// Brief: Master Arm Standby
FUNCTION_BLOCK PUBLIC FB_StateCtrlPanelReady EXTENDS FB_SlaveArmCtrlBase
VAR_INPUT
END_VAR
VAR_OUTPUT
END_VAR
VAR
END_VAR

END_FUNCTION_BLOCK

(* stored: Version 1.1.0.1, ProductVersion 3.1.4024.12
   POU FB_StateCtrlPanelReady: Id {f4ef749e-f294-45ac-8079-35edcc11796e}, SpecialFunc None *)
